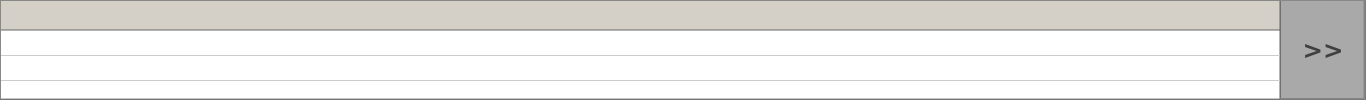
VISUALIZATION PH_Bottom  // 1366x100
VAR_IN_OUT
	bReset 									: BOOL;
	arrEventVisu							: ARRAY [1..GVL_EHS.diNoOfEvents] OF ST_EventHistoricalSimple;	 
END_VAR
    Table (0,0 1280x100), data array: GVL_EHS.arrEventVisu
        p3854506369: GVL_EHS.arrEventVisu[INDEX].dwID
        p505689113: Date End
        p1218418051: GVL_EHS.arrEventVisu[INDEX].dtDateEnd
        p2237128397: Date Begin
        p3723444502: GVL_EHS.arrEventVisu[INDEX].dtDateBegin
        p4092479075: Param
        p2170511999: GVL_EHS.arrEventVisu[INDEX].dwParam
        p511219082: Class
        p1892666644: GVL_EHS.arrEventVisu[INDEX].dwClass
        p1755163831: Message
        p338671338: GVL_EHS.arrEventVisu[INDEX].wsMessage
        Columns.Column.[2].Template: GVL_EHS.arrEventVisu[INDEX].dwColor
        Columns.Column.[0].Template: GVL_EHS.arrEventVisu[INDEX].dwColor
        Columns.Column.[1].Template: GVL_EHS.arrEventVisu[INDEX].dwColor
        Columns.Column.[4].Template: GVL_EHS.arrEventVisu[INDEX].dwColor
        Columns.Column.[3].Template: GVL_EHS.arrEventVisu[INDEX].dwColor
        Columns.Column.[5].Template: GVL_EHS.arrEventVisu[INDEX].dwColor
    Button (1280,0 86x100), ">>"
        OnMouseDown: execute { GVL_HMI.iFrameNumber:=1; GVL_HMI.bMenu:=FALSE; }
END_VISUALIZATION

(* stored: Version 1.1.0.1, ProductVersion 3.1.4024.3
   Visu PH_Bottom: Id {725c07d8-7b83-4f8a-9823-cc0386cb4b97} *)
